{attribute 'Tc2GvlVarNames'}
VAR_GLOBAL
	
	(* Ping *)
	bUseTasterPing				:BOOL := FALSE;			(* Schaltet den Dauerping für die Taster ein *)	(* Wird noch nicht verwendet, da es nicht so zuverlässig Funktioniert *)
	bUseRelaisPing				:BOOL := FALSE;			(* Schaltet den Dauerping für die Relais ein *)	(* Wird noch nicht verwendet, da es nicht so zuverlässig Funktioniert *)
	
	cTimePingTimeRelais			:TIME := T#10S;			(* Ping Intervallzeit *)
	cTimeReceiveTimeoutRelais	:TIME := T#200MS;		(* Ping Empfangs Timeout *)
	
	cTimePingTimeTaster			:TIME := T#5M;			(* Ping Intervallzeit *)	(* Vorerst auf 5min gestellt, da die Taster Automatisch senden (Helligkeit/Luftfeuchtigkeit/Temp usw. *)
	cTimeReceiveTimeoutTaster	:TIME := T#200MS;		(* Ping Empfangs Timeout *)
	
	cMaxPingTry					:INT :=	5;				(* Anzahl der Pingversuche *)
	
END_VAR

(* stored: Version 1.1.0.1, ProductVersion 3.1.4024.12
   GVL GVL_HausBus_Parameter_1: Id {0a07316c-bf5f-4da2-b07e-6241ad791d0b} *)
